FUNCTION F_EcDeviceTimeStampToTime : TIME
VAR_INPUT
	nDeviceTimeStamp : ULINT;
END_VAR
VAR
	fDevieTimeStamp : LREAL;
END_VAR

fDevieTimeStamp := ULINT_TO_LREAL(nDeviceTimeStamp) / 1E6; 		// ns to ms
F_EcDeviceTimeStampToTime := LREAL_TO_TIME(fDevieTimeStamp);	// ms to time

END_FUNCTION

(* stored: Version 1.1.0.1, ProductVersion 3.1.4024.12
   POU F_EcDeviceTimeStampToTime: Id {f18413ab-7b27-43ac-9ece-1ef07923db69}, SpecialFunc None *)
